{attribute 'linkalways'} 
{attribute 'no_explicit_call' := 'This FB is a CLASS and must be accessed using methods or properties'}
{attribute 'enable_dynamic_creation'}
FUNCTION_BLOCK ABSTRACT Error EXTENDS Disposable IMPLEMENTS I_Error
VAR
END_VAR

METHOD PUBLIC Accept
VAR_INPUT
	Visitor : I_ErrorVisitor;
END_VAR
Visitor.VisitError(THIS^);
END_METHOD

PROPERTY PUBLIC ABSTRACT ErrorType : T_MAXSTRING
GET
END_GET
END_PROPERTY

METHOD PUBLIC IsSameAs : BOOL
VAR_INPUT
	Error : I_Error;
END_VAR
IF Error = 0 THEN
	RETURN;
END_IF

IF Error.ErrorType <> THIS^.ErrorType THEN
	RETURN;
END_IF

IsSameAs := TRUE;
END_METHOD

PROPERTY PUBLIC ABSTRACT Message : T_MAXSTRING
GET
END_GET
END_PROPERTY

METHOD PROTECTED OnSerialize
VAR_INPUT
	Serializer : I_Serializer;
END_VAR
END_METHOD

METHOD PUBLIC SerializeWith
VAR_INPUT
	Serializer : I_Serializer;
END_VAR
Serializer.StartObject();
Serializer.AddKeyString('errorType',ErrorType);
Serializer.AddKeyString('message',Message);
OnSerialize(Serializer);
Serializer.EndObject();
END_METHOD

END_FUNCTION_BLOCK

(* stored: Version 1.1.0.1, ProductVersion 3.1.4024.12
   POU Error: Id {7c55cd79-4747-018f-312f-869bc7e0f09a}, SpecialFunc None
   Folder Protected: Id {c13f1263-be0b-02bd-016c-016a337233da}
   Method Accept: Id {fef303be-3cc4-0248-280b-0a344804d08c}
   Property ErrorType: Id {5854729a-7d9b-01f6-22a5-51325658dc5f}
   Get Get: Id {ace55bdd-3310-0f83-038f-b9582177b9b5}
   Method IsSameAs: Id {f504f489-f2c1-035a-208c-cda66e566b41}
   Property Message: Id {abe30e40-2d6e-03b7-2b21-bb7337aadbd9}
   Get Get: Id {95155e29-8281-0bd0-1dd2-bab04737c95b}
   Method OnSerialize: Id {cb0b2354-a014-04ff-3bcf-6e98b9d20f11}
   Method SerializeWith: Id {598303df-8e61-0b5a-2cea-15656226d0b2} *)
